FUNCTION_BLOCK FileSink IMPLEMENTS ITcoLogSink
VAR_INPUT
END_VAR
VAR_OUTPUT
END_VAR
VAR
	_filePath		: STRING(255);
END_VAR

METHOD Emit : BOOL
VAR_INPUT
	LogEvent	: REFERENCE TO LogEvent;
END_VAR
// Write to file writer buffer


// e.g. use sample of benhar-dev
// https://github.com/benhar-dev/tc3-data-logger
END_METHOD

PROPERTY PUBLIC FilePath : STRING(255)
GET
FilePath := _filePath;
END_GET
SET
_filePath := FilePath;
END_SET
END_PROPERTY

END_FUNCTION_BLOCK

(* stored: Version 1.1.0.1, ProductVersion 3.1.4024.9
   POU FileSink: Id {9a0372bc-f0f0-04ef-2fa5-e601c4eee8b0}, SpecialFunc None
   Method Emit: Id {ebf12252-d03b-0b9c-3ff6-e03360967b56}
   Property FilePath: Id {389a9893-b016-0ad1-01d7-a2ef620a43da}
   Get Get: Id {8e28db3d-55bd-0169-07ed-18d48d5279c4}
   Set Set: Id {b068213b-984a-0feb-380a-914bc3bbd9d0} *)
